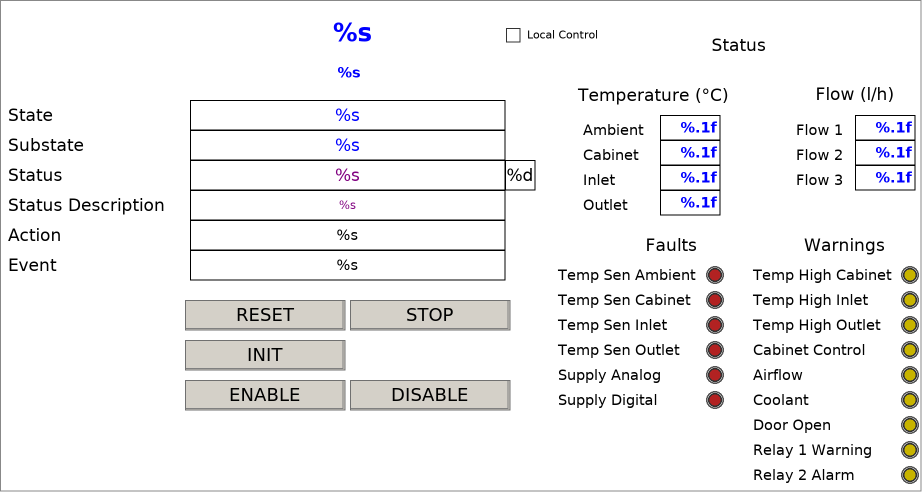
VISUALIZATION GUI_TEMPLATE_CCC  // 922x492
VAR_IN_OUT
	m_Instance:	FB_CCC;
END_VAR
    Rectangle (190,100 315x30), "%s", text variable: m_Instance.stat.sState
    Rectangle (190,130 315x30), "%s", text variable: m_Instance.stat.sSubstate
    Button (185,300 160x30), "RESET", input disabled if: (m_Instance.stat.bLocal = FALSE) <> 0
        OnMouseClick: execute { m_Instance.ctrl.nCommand := E_RS_COMMAND.RESET; m_Instance.ctrl.bExecute := TRUE; }
    Button (185,340 160x30), "INIT", input disabled if: (m_Instance.stat.bLocal = FALSE) <> 0
        OnMouseClick: execute { m_Instance.ctrl.nCommand := E_RS_COMMAND.INIT; m_Instance.ctrl.bExecute := TRUE; }
    Button (350,300 160x30), "STOP", input disabled if: (m_Instance.stat.bLocal = FALSE) <> 0
        OnMouseClick: execute { m_Instance.ctrl.nCommand := E_RS_COMMAND.STOP; m_Instance.ctrl.bExecute := TRUE; }
    Button (185,380 160x30), "ENABLE", input disabled if: (m_Instance.stat.bLocal = FALSE) <> 0
        OnMouseClick: execute { m_Instance.ctrl.nCommand := E_RS_COMMAND.ENABLE; m_Instance.ctrl.bExecute := TRUE; }
    Button (350,380 160x30), "DISABLE", input disabled if: (m_Instance.stat.bLocal = FALSE) <> 0
        OnMouseClick: execute { m_Instance.ctrl.nCommand := E_RS_COMMAND.DISABLE; m_Instance.ctrl.bExecute := TRUE; }
    Rectangle (5,100 180x30), "State"
    Rectangle (5,130 180x30), "Substate"
    Rectangle (190,160 315x30), "%s", text variable: m_Instance.stat.sStatus
    Rectangle (190,190 315x30), "%s", text variable: m_Instance.stat.sErrorText
    Rectangle (5,160 180x30), "Status"
    Rectangle (5,190 180x30), "Status Description"
    Rectangle (190,220 315x30), "%s", text variable: m_Instance.stat.sActionDesc
    Rectangle (190,250 315x30), "%s", text variable: m_Instance.stat.sEventDesc
    Rectangle (5,220 180x30), "Action"
    Rectangle (5,250 180x30), "Event"
    Rectangle (266,15 173x35), "%s", text variable: m_Instance.in_sName
    Checkbox (504,20 116x30), "Local Control", variable: m_Instance.stat.bLocal
    Rectangle (693,30 92x30), "Status"
    Rectangle (505,160 30x30), "%d", text variable: m_Instance.stat.nStatus
    Rectangle (569,80 169x30), "Temperature (°C)"
    Rectangle (806,79 98x30), "Flow (l/h)"
    Rectangle (580,115 70x30), "Ambient"
    Rectangle (580,140 70x30), "Cabinet"
    Rectangle (580,165 70x30), "Inlet"
    Rectangle (580,190 70x30), "Outlet"
    Rectangle (660,115 60x25), "%.1f", text variable: m_Instance.stat.lrTemp_ambient
    Rectangle (660,140 60x25), "%.1f", text variable: m_Instance.stat.lrTemp_cabinet
    Rectangle (660,165 60x25), "%.1f", text variable: m_Instance.stat.lrTemp_inlet
    Rectangle (660,190 60x25), "%.1f", text variable: m_Instance.stat.lrTemp_outlet
    Rectangle (855,115 60x25), "%.1f", text variable: m_Instance.stat.lrFlow_1
    Rectangle (781,115 65x30), "Flow 1"
    Rectangle (781,140 65x30), "Flow 2"
    Rectangle (855,140 60x25), "%.1f", text variable: m_Instance.stat.lrFlow_2
    Rectangle (781,165 65x30), "Flow 3"
    Rectangle (855,165 60x25), "%.1f", text variable: m_Instance.stat.lrFlow_3
    Rectangle (605,230 133x30), "Faults"
    Rectangle (555,260 150x30), "Temp Sen Ambient"
    Lamp1 (705,265 20x20), variable: m_Instance.stat.bFault_temp_sensor_ambient, style: Lamp-Lamp1-Red
    Rectangle (555,285 150x30), "Temp Sen Cabinet"
    Lamp1 (705,290 20x20), variable: m_Instance.stat.bFault_temp_sensor_cabinet, style: Lamp-Lamp1-Red
    Rectangle (555,310 150x30), "Temp Sen Inlet"
    Lamp1 (705,315 20x20), variable: m_Instance.stat.bFault_temp_sensor_inlet, style: Lamp-Lamp1-Red
    Rectangle (555,335 150x30), "Temp Sen Outlet"
    Lamp1 (705,340 20x20), variable: m_Instance.stat.bFault_temp_sensor_outlet, style: Lamp-Lamp1-Red
    Rectangle (555,360 150x30), "Supply Analog"
    Lamp1 (705,365 20x20), variable: m_Instance.stat.bFault_analog_supply, style: Lamp-Lamp1-Red
    Rectangle (555,385 150x30), "Supply Digital"
    Lamp1 (705,390 20x20), variable: m_Instance.stat.bFault_digital_supply, style: Lamp-Lamp1-Red
    Rectangle (778,230 133x30), "Warnings"
    Rectangle (750,260 150x30), "Temp High Cabinet"
    Lamp1 (900,265 20x20), variable: m_Instance.stat.bWarn_cabinet_high, style: Lamp-Lamp1-Yellow
    Rectangle (750,335 150x30), "Cabinet Control"
    Lamp1 (900,340 20x20), variable: m_Instance.stat.bWarn_cabinet_no_control, style: Lamp-Lamp1-Yellow
    Rectangle (750,310 150x30), "Temp High Outlet"
    Lamp1 (900,315 20x20), variable: m_Instance.stat.bWarn_outlet_high, style: Lamp-Lamp1-Yellow
    Rectangle (750,285 150x30), "Temp High Inlet"
    Lamp1 (900,290 20x20), variable: m_Instance.stat.bWarn_inlet_high, style: Lamp-Lamp1-Yellow
    Rectangle (750,360 150x30), "Airflow"
    Lamp1 (900,365 20x20), variable: m_Instance.stat.bWarn_airflow_insufficient, style: Lamp-Lamp1-Yellow
    Rectangle (750,385 150x30), "Coolant"
    Lamp1 (900,390 20x20), variable: m_Instance.stat.bWarn_coolant_insufficient, style: Lamp-Lamp1-Yellow
    Rectangle (750,410 150x30), "Door Open"
    Lamp1 (900,415 20x20), variable: m_Instance.stat.bWarn_door_open, style: Lamp-Lamp1-Yellow
    Rectangle (750,435 150x30), "Relay 1 Warning"
    Lamp1 (900,440 20x20), variable: m_Instance.stat.bWarn_relay1_warning, style: Lamp-Lamp1-Yellow
    Rectangle (750,460 150x30), "Relay 2 Alarm"
    Lamp1 (900,465 20x20), variable: m_Instance.stat.bWarn_relay2_alarm, style: Lamp-Lamp1-Yellow
    Rectangle (184,60 330x25), "%s", text variable: m_Instance.stat.sDeviceID
END_VISUALIZATION

(* stored: Version 1.1.0.1, ProductVersion 3.1.4022.16
   Visu GUI_TEMPLATE_CCC: Id {58f7adab-bf2b-466d-bc90-b3570e944a44} *)
